PROGRAM SFC
VAR
	Run: BOOL;
	After15s: BOOL;
	Finished: BOOL;
	SteamIn: BOOL;
	Drain: BOOL;
	WaterIn: BOOL;
	GlycolIn: BOOL;
	GlycolOut: BOOL;
	Temp: REAL;
	FlushTimer: TON;
	Temp_GE_70: BOOL;
	Temp_LE_4: BOOL;
	Temp_LT_20: BOOL;
END_VAR

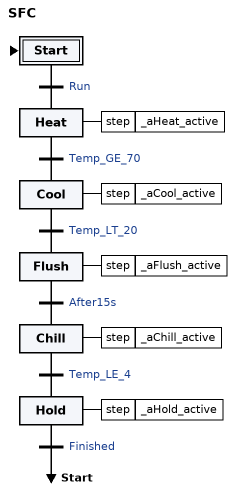
INITIAL_STEP Start:
END_STEP
TRANSITION FROM Start TO Heat
    := Run;
END_TRANSITION
STEP Heat:
    _aHeat_active(N);  // step action
END_STEP
TRANSITION FROM Heat TO Cool
    := Temp_GE_70;
END_TRANSITION
STEP Cool:
    _aCool_active(N);  // step action
END_STEP
TRANSITION FROM Cool TO Flush
    := Temp_LT_20;
END_TRANSITION
STEP Flush:
    _aFlush_active(N);  // step action
END_STEP
TRANSITION FROM Flush TO Chill
    := After15s;
END_TRANSITION
STEP Chill:
    _aChill_active(N);  // step action
END_STEP
TRANSITION FROM Chill TO Hold
    := Temp_LE_4;
END_TRANSITION
STEP Hold:
    _aHold_active(N);  // step action
END_STEP
TRANSITION FROM Hold TO Start
    := Finished;
END_TRANSITION

ACTION _aChill_active:
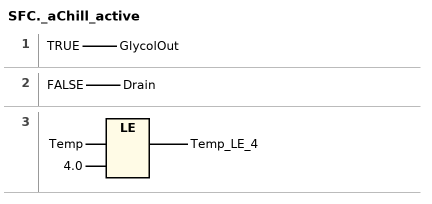
// NETWORK 1
GlycolOut := TRUE;

// NETWORK 2
Drain := FALSE;

// NETWORK 3
Temp_LE_4 := Temp <= 4.0;
END_ACTION

ACTION _aCool_active:
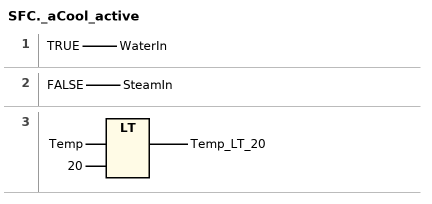
// NETWORK 1
WaterIn := TRUE;

// NETWORK 2
SteamIn := FALSE;

// NETWORK 3
Temp_LT_20 := Temp < 20;
END_ACTION

ACTION _aFlush_active:
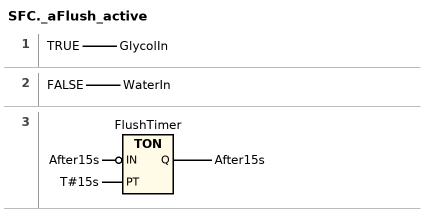
// NETWORK 1
GlycolIn := TRUE;

// NETWORK 2
WaterIn := FALSE;

// NETWORK 3
FlushTimer(IN := NOT After15s, PT := T#15s); // TON
After15s := FlushTimer.Q;
END_ACTION

ACTION _aHeat_active:
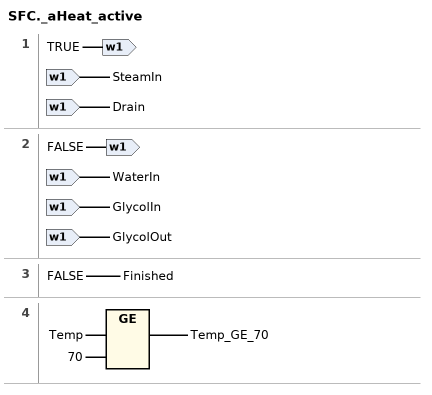
// NETWORK 1
SteamIn := TRUE;
Drain := TRUE;

// NETWORK 2
WaterIn := FALSE;
GlycolIn := FALSE;
GlycolOut := FALSE;

// NETWORK 3
Finished := FALSE;

// NETWORK 4
Temp_GE_70 := Temp >= 70;
END_ACTION

ACTION _aHold_active:
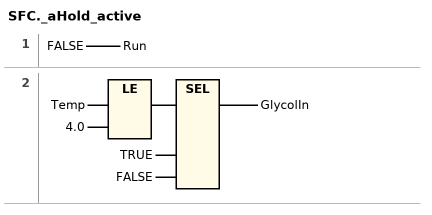
// NETWORK 1
Run := FALSE;

// NETWORK 2
GlycolIn := SEL(Temp <= 4.0, TRUE, FALSE);
END_ACTION

END_PROGRAM

(* stored: Version 1.1.0.1, ProductVersion 3.1.4024.12
   POU SFC: Id {0d703742-8800-4c6f-96df-ce43e91e7df4}, SpecialFunc None
   Action _aChill_active: Id {c5d7e1c7-4ce6-4887-9553-a1356f52e0ff}
   Action _aCool_active: Id {e1626dfe-7856-4f03-a51a-cd9ad1579a65}
   Action _aFlush_active: Id {708affcb-828e-43bc-b136-ee8adbd84df5}
   Action _aHeat_active: Id {a93ebbff-70d0-42d1-a578-e1af984cad58}
   Action _aHold_active: Id {307e74d7-d3af-445a-81ac-9b84a9ebf99b} *)
